# EPICS IOC start-up script: iocs/smarActIOC/iocBoot/iocSmarAct/smaractmcs2.iocsh
drvAsynIPPortConfigure("MCS2_ETH", "192.168.1.200:55551", 0, 0, 0)

dbLoadRecords("$(ASYN)/db/asynRecord.db", "P=Test{MC:T}, R=Asyn, PORT=MCS2_ETH, ADDR=0, OMAX=256, IMAX=256")

# PORT, MCS_PORT, number of axes, active poll period (ms), idle poll period (ms)
MCS2CreateController("MCS2", "MCS2_ETH", 3, 100, 100)
MCS2CreateAxis("MCS2",0)

dbLoadTemplate "motor.substitutions.smaractmcs2"

#asynSetTraceMask("MCS2", 0, 0x4)
#asynSetTraceIOMask("MCS2", -1, 0x8)
